// TwinCAT 3 PLC project SIM
// ProgramVersion: 3.1.4020.5
// libraries:
//   Tc2_Standard, * (Beckhoff Automation GmbH)
//   Tc2_System, * (Beckhoff Automation GmbH)
//   Tc3_Module, * (Beckhoff Automation GmbH)
//   Vacuum System Simulator Library, * (SLAC)
// project tree:
//   GVLs/ GVL_IO.TcGVL, GVL_SimDevices.TcGVL
//   / PlcTaskSim.TcTTO
//   POUs/ MAIN.TcPOU, OverridePressure.TcPOU, SoftIO.TcPOU
// (motion and I/O tree: see PLC project test)
// real-time tasks:
//   TASK PlcTask: cycle T#10ms, priority 20, ADS port 350
//   TASK SimTask: cycle T#10ms, priority 1, ADS port 351
//   TASK VacTask: cycle T#10ms, priority 2, ADS port 352
// variable links:
//   SIM/SIM Instance <-> test/test Instance
//     PlcTaskSim Inputs/GVL_SimDevices.S_FEE_GCC_03.i_xHvOn <-> PlcTask Outputs/GVL_Devices.FEE_GCC_03.q_xHV_DIS
//     PlcTaskSim Inputs/GVL_SimDevices.S_FEE_GCC_04.i_xHvOn <-> PlcTask Outputs/GVL_Devices.FEE_GCC_04.q_xHV_DIS
//     PlcTaskSim Inputs/GVL_SimDevices.S_FEE_KMONO_GCC_01.i_xHvOn <-> PlcTask Outputs/GVL_Devices.FEE_KMONO_GCC_01.q_xHV_DIS
//     PlcTaskSim Inputs/GVL_SimDevices.S_FEE_KMONO_PIP_01.xOn <-> PlcTask Outputs/GVL_Devices.FEE_KMONO_PIP_01.q_xHVEna_DO
//     PlcTaskSim Inputs/GVL_SimDevices.S_FEE_M1L_PIP_01.xOn <-> PlcTask Outputs/GVL_Devices.FEE_M1L_PIP_01.q_xHVEna_DO
//     PlcTaskSim Inputs/GVL_SimDevices.S_FEE_MIL_GCC_02.i_xHvOn <-> PlcTask Outputs/GVL_Devices.FEE_M1L_GCC_01.q_xHV_DIS
//     PlcTaskSim Inputs/GVL_SimDevices.S_FEE_PIP_02.xOn <-> PlcTask Outputs/GVL_Devices.FEE_PIP_02.q_xHVEna_DO
//     PlcTaskSim Inputs/GVL_SimDevices.S_FEE_PIP_03.xOn <-> PlcTask Outputs/GVL_Devices.FEE_PIP_03.q_xHVEna_DO
//     PlcTaskSim Inputs/GVL_SimDevices.S_FEE_VGC_02.i_xSol <-> PlcTask Outputs/GVL_Devices.FEE_VGC_02.q_xOPN_DO
//     PlcTaskSim Inputs/GVL_SimDevices.S_FEE_VGC_03.i_xSol <-> PlcTask Outputs/GVL_Devices.FEE_VGC_03.q_xOPN_DO
//     PlcTaskSim Inputs/GVL_SimDevices.S_FEE_VGC_04.i_xSol <-> PlcTask Outputs/GVL_Devices.FEE_VGC_04.q_xOPN_DO
//     PlcTaskSim Inputs/GVL_SimDevices.VGC_1.i_xSol <-> PlcTask Outputs/PRG_VLS.VGC_1.q_xOPN_DO
//     PlcTaskSim Inputs/GVL_SimDevices.VGC_W.i_xSol <-> PlcTask Outputs/PRG_VLS.VGC_W.q_xCLS_DO
//     PlcTaskSim Outputs/GVL_SimDevices.S_FEE_GCC_03.q_DisActive <-> PlcTask Inputs/GVL_Devices.FEE_GCC_03.i_xDisc_Active
//     PlcTaskSim Outputs/GVL_SimDevices.S_FEE_GCC_04.q_DisActive <-> PlcTask Inputs/GVL_Devices.FEE_GCC_04.i_xDisc_Active
//     PlcTaskSim Outputs/GVL_SimDevices.S_FEE_GCC_03.q_iRawPress <-> PlcTask Inputs/GVL_Devices.FEE_GCC_03.i_iPRESS_R
//     PlcTaskSim Outputs/GVL_SimDevices.S_FEE_GCC_04.q_iRawPress <-> PlcTask Inputs/GVL_Devices.FEE_GCC_04.i_iPRESS_R
//     PlcTaskSim Outputs/GVL_SimDevices.S_FEE_GCC_03.q_iRawPress <-> PlcTask Inputs/PRG_VLS.DS_GCC.i_iPRESS_R
//     PlcTaskSim Outputs/GVL_SimDevices.S_FEE_GCC_03.q_xHVOn <-> PlcTask Inputs/GVL_Devices.FEE_GCC_03.i_xHV_ON
//     PlcTaskSim Outputs/GVL_SimDevices.S_FEE_GCC_04.q_xHVOn <-> PlcTask Inputs/GVL_Devices.FEE_GCC_04.i_xHV_ON
//     PlcTaskSim Outputs/GVL_SimDevices.S_FEE_GPI_03.q_iRawPress <-> PlcTask Inputs/GVL_Devices.FEE_GPI_03.i_iPRESS_R
//     PlcTaskSim Outputs/GVL_SimDevices.S_FEE_GPI_04.q_iRawPress <-> PlcTask Inputs/GVL_Devices.FEE_GPI_04.i_iPRESS_R
//     PlcTaskSim Outputs/GVL_SimDevices.S_FEE_GPI_03.q_iRawPress <-> PlcTask Inputs/PRG_VLS.DS_GPI.i_iPRESS_R
//     PlcTaskSim Outputs/GVL_SimDevices.S_FEE_KMONO_GCC_01.q_DisActive <-> PlcTask Inputs/GVL_Devices.FEE_KMONO_GCC_01.i_xDisc_Active
//     PlcTaskSim Outputs/GVL_SimDevices.S_FEE_KMONO_GCC_01.q_iRawPress <-> PlcTask Inputs/GVL_Devices.FEE_KMONO_GCC_01.i_iPRESS_R
//     PlcTaskSim Outputs/GVL_SimDevices.S_FEE_KMONO_GCC_01.q_iRawPress <-> PlcTask Inputs/PRG_VLS.US_GCC.i_iPRESS_R
//     PlcTaskSim Outputs/GVL_SimDevices.S_FEE_KMONO_GCC_01.q_xHVOn <-> PlcTask Inputs/GVL_Devices.FEE_KMONO_GCC_01.i_xHV_ON
//     PlcTaskSim Outputs/GVL_SimDevices.S_FEE_KMONO_GPI_01.q_iRawPress <-> PlcTask Inputs/GVL_Devices.FEE_KMONO_GPI_01.i_iPRESS_R
//     PlcTaskSim Outputs/GVL_SimDevices.S_FEE_KMONO_GPI_01.q_iRawPress <-> PlcTask Inputs/PRG_VLS.US_GPI.i_iPRESS_R
//     PlcTaskSim Outputs/GVL_SimDevices.S_FEE_M1L_GPI_02.q_iRawPress <-> PlcTask Inputs/GVL_Devices.FEE_M1L_GPI_01.i_iPRESS_R
//     PlcTaskSim Outputs/GVL_SimDevices.S_FEE_MIL_GCC_02.q_DisActive <-> PlcTask Inputs/GVL_Devices.FEE_M1L_GCC_01.i_xDisc_Active
//     PlcTaskSim Outputs/GVL_SimDevices.S_FEE_MIL_GCC_02.q_iRawPress <-> PlcTask Inputs/GVL_Devices.FEE_M1L_GCC_01.i_iPRESS_R
//     PlcTaskSim Outputs/GVL_SimDevices.S_FEE_MIL_GCC_02.q_xHVOn <-> PlcTask Inputs/GVL_Devices.FEE_M1L_GCC_01.i_xHV_ON
//     PlcTaskSim Outputs/GVL_SimDevices.S_FEE_VGC_02.q_xClsLS <-> PlcTask Inputs/GVL_Devices.FEE_VGC_02.i_xClsLS
//     PlcTaskSim Outputs/GVL_SimDevices.S_FEE_VGC_03.q_xClsLS <-> PlcTask Inputs/GVL_Devices.FEE_VGC_03.i_xClsLS
//     PlcTaskSim Outputs/GVL_SimDevices.S_FEE_VGC_04.q_xClsLS <-> PlcTask Inputs/GVL_Devices.FEE_VGC_04.i_xClsLS
//     PlcTaskSim Outputs/GVL_SimDevices.S_FEE_VGC_02.q_xOpnLS <-> PlcTask Inputs/GVL_Devices.FEE_VGC_02.i_xOpnLS
//     PlcTaskSim Outputs/GVL_SimDevices.S_FEE_VGC_03.q_xOpnLS <-> PlcTask Inputs/GVL_Devices.FEE_VGC_03.i_xOpnLS
//     PlcTaskSim Outputs/GVL_SimDevices.S_FEE_VGC_04.q_xOpnLS <-> PlcTask Inputs/GVL_Devices.FEE_VGC_04.i_xOpnLS
//     PlcTaskSim Outputs/GVL_SimDevices.VGC_1.q_xClsLS <-> PlcTask Inputs/PRG_VLS.VGC_1.i_xClsLS
//     PlcTaskSim Outputs/GVL_SimDevices.VGC_1.q_xOpnLS <-> PlcTask Inputs/PRG_VLS.VGC_1.i_xOpnLS
//     PlcTaskSim Outputs/GVL_SimDevices.VGC_W.q_xClsLS <-> PlcTask Inputs/PRG_VLS.VGC_W.i_xClsLS
//     PlcTaskSim Outputs/GVL_SimDevices.VGC_W.q_xOpnLS <-> PlcTask Inputs/PRG_VLS.VGC_W.i_xOpnLS

CONFIGURATION SIM
    RESOURCE PLC ON TwinCAT3
        TASK PlcTaskSim(INTERVAL := T#10ms, PRIORITY := 1);
        PROGRAM MAIN WITH PlcTaskSim : MAIN;
    END_RESOURCE
END_CONFIGURATION

// ---- GVLs/GVL_IO.TcGVL
VAR_GLOBAL
	
(*pumps*)
(*
S_FEE_KMONO_PIP_01_xON AT%I*:BOOL;
S_FEE_PIP_02_xON AT%I*:BOOL;
S_FEE_M1L_PIP_01_xON AT%I*:BOOL;
S_FEE_PIP_03_xON AT%I*:BOOL;*)


(*Valves*)

END_VAR

// ---- GVLs/GVL_SimDevices.TcGVL
VAR_GLOBAL
	Global_Leak	: REAL := 0;
	Global_Pressure : REAL := 0.0079;
	New_Pressure : REAL := 22.0; //Torr
	Global_OverridePressure	: BOOL := FALSE;//initially set to be false
(* Volumes *)
	
	//-1
	stVl_Start	:	ST_Volume:=(
		rPressure := Global_Pressure,
		rVolume := 1E3,
		rVLeak	:= Global_Leak
		);
		
	//0) KMONO
	stVl_KMONO	:	ST_Volume:=(
		rPressure := Global_Pressure,
		rVolume := 1E3,
		rVLeak	:= Global_Leak
		);
	
	//1) M1L0
	stVl_M1L0	:	ST_Volume:=(
		rPressure := Global_Pressure,
		rVolume := 1E3,
		rVLeak	:= Global_Leak
		);
		
		//1) End
	stVl_End	:	ST_Volume:=(
		rPressure := Global_Pressure,
		rVolume := 1E3,
		rVLeak	:= Global_Leak
		);
		
(*Valves*)
	VGC_1 : ST_VacuumValve:=(
		q_xClsLS := TRUE,
		q_xOpnLS := FALSE
	);
	VGC_2 : ST_VacuumValve:=(
		q_xClsLS := TRUE,
		q_xOpnLS := FALSE
	);
	VGC_W : ST_VacuumValve:=(
		q_xClsLS := TRUE,
		q_xOpnLS := FALSE
	);
	
	S_FEE_VGC_02 : ST_VacuumValve:=(
		q_xClsLS := TRUE,
		q_xOpnLS := FALSE
	);
	
	S_FEE_VGC_03 : ST_VacuumValve:=(
		q_xClsLS := TRUE,
		q_xOpnLS := FALSE
	);
	
	S_FEE_VGC_04 : ST_VacuumValve:=(
		q_xClsLS := TRUE,
		q_xOpnLS := FALSE
	);

(*Gauges*)
	S_FEE_KMONO_GPI_01 : ST_MKS_275 :=(
		q_xGaugeConnected := TRUE
	);
	S_FEE_KMONO_GCC_01 : ST_MKS_500 :=(
		q_xGaugeConnected := TRUE
	);
	S_FEE_GPI_03 : ST_MKS_275 :=(
		q_xGaugeConnected := TRUE
	);
	S_FEE_GCC_03 : ST_MKS_500 :=(
		q_xGaugeConnected := TRUE
	);
	S_FEE_M1L_GPI_02 : ST_MKS_275 :=(
		q_xGaugeConnected := TRUE
	);
	S_FEE_MIL_GCC_02 : ST_MKS_500 :=(
		q_xGaugeConnected := TRUE
	);
	S_FEE_GPI_04 : ST_MKS_275 :=(
		q_xGaugeConnected := TRUE
	);
	S_FEE_GCC_04 : ST_MKS_500 :=(
		q_xGaugeConnected := TRUE
	);
	
(*ION Pumps*)
	S_FEE_KMONO_PIP_01 : ST_GAM_PIP; 
	S_FEE_PIP_02 : ST_GAM_PIP; 
	S_FEE_M1L_PIP_01 : ST_GAM_PIP; 
	S_FEE_PIP_03 : ST_GAM_PIP; 

(*Turbo and VRC*)
	
END_VAR

// ---- POUs/MAIN.TcPOU
PROGRAM MAIN
VAR
	
	(*Valves*)
	fb_VGC_1 : FB_VacuumValve;
	fb_VGC_2 : FB_VacuumValve;
	fb_VGC_W : FB_VacuumValve_Vent; //NO valve


	(*Valves*)
	fb_VGC_02 : FB_VacuumValve;
	fb_VGC_03 : FB_VacuumValve;
	fb_VGC_04 : FB_VacuumValve;
	
	
	(*Gauges*)
	fbMKS500_VGCC_KMONO_01	:	FB_MKS_500;
	fbMKS500_VGCC_03	:	FB_MKS_500;
	fbMKS500_VGCC_M1L_01	:	FB_MKS_500;
	fbMKS500_VGCC_04	:	FB_MKS_500;
	
	fbMKS500_VGPI_KMONO_01	:	FB_MKS_275;
	fbMKS500_VGPI_03	:	FB_MKS_275;
	fbMKS500_VGPI_M1L_01	:	FB_MKS_275;
	fbMKS500_VGPI_04	:	FB_MKS_275;
	
	(*Ion Pumps*)
	fb_PIP_KMONO_01	:	FB_GAM_PIP;
	fb_PIP_02	:	FB_GAM_PIP;
	fb_PIP_M1L_01	:	FB_GAM_PIP;
	fb_PIP_03	:	FB_GAM_PIP;
	
	
END_VAR

OverridePressure();

(*Valves*)

fb_VGC_1(stAVol:=stVl_Start , 
	stBVol:= stVl_KMONO,
	stValve:= VGC_1
	);

fb_VGC_2(stAVol:=stVl_Start , 
	stBVol:= stVl_KMONO,
	stValve:= VGC_2
	);
fb_VGC_W(stAVol:=stVl_Start , 
	stBVol:= stVl_KMONO,
	stValve:= VGC_W
	);



fb_VGC_02(stAVol:=stVl_Start , 
	stBVol:= stVl_KMONO,
	stValve:= S_FEE_VGC_02
	);
	
fb_VGC_03(stAVol:= stVl_KMONO, 
	stBVol:= stVl_M1L0,
	stValve:= S_FEE_VGC_03
	);	
	
fb_VGC_04(stAVol:= stVl_M1L0, 
	stBVol:= stVl_End,
	stValve:= S_FEE_VGC_04
	);	
	

(*Gauges*)
fbMKS500_VGCC_KMONO_01(stVolume := stVl_KMONO, stGauge := S_FEE_KMONO_GCC_01);
fbMKS500_VGPI_KMONO_01(stVolume := stVl_KMONO, stGauge := S_FEE_KMONO_GPI_01);

fbMKS500_VGCC_03(stVolume := stVl_KMONO, stGauge := S_FEE_GCC_03);
fbMKS500_VGPI_03(stVolume := stVl_KMONO, stGauge := S_FEE_GPI_03);

fbMKS500_VGCC_M1L_01(stVolume := stVl_M1L0, stGauge := S_FEE_MIL_GCC_02);
fbMKS500_VGPI_M1L_01(stVolume := stVl_M1L0, stGauge := S_FEE_M1L_GPI_02);

fbMKS500_VGCC_04(stVolume := stVl_M1L0, stGauge := S_FEE_GCC_04);
fbMKS500_VGPI_04(stVolume := stVl_M1L0, stGauge := S_FEE_GPI_04);


(*Ion Pumps*)
fb_PIP_KMONO_01(stVolume:= stVl_KMONO, stPip:= S_FEE_KMONO_PIP_01);
fb_PIP_02(stVolume:= stVl_KMONO, stPip:= S_FEE_PIP_02);
fb_PIP_M1L_01(stVolume:= stVl_M1L0, stPip:= S_FEE_M1L_PIP_01);
fb_PIP_03(stVolume:= stVl_M1L0, stPip:= S_FEE_PIP_03);

END_PROGRAM

// ---- POUs/OverridePressure.TcPOU
PROGRAM OverridePressure
VAR
	fb_SetPressure : FB_SetChamberPressure; 
END_VAR

fb_SetPressure(chamber := stVl_KMono, rNewPressure := New_Pressure, Override:= Global_OverridePressure);

END_PROGRAM

// ---- POUs/SoftIO.TcPOU
PROGRAM SoftIO
VAR
END_VAR

(*S_FEE_KMONO_PIP_01.xOn := S_FEE_KMONO_PIP_01_xON;
S_FEE_PIP_02.xOn := S_FEE_PIP_02_xON ;
S_FEE_M1L_PIP_01.xOn := S_FEE_M1L_PIP_01_xON;
S_FEE_PIP_03.xOn := S_FEE_PIP_03_xON;*)

END_PROGRAM
